{attribute 'linkalways'} 
{attribute 'no_explicit_call' := 'This FB is a CLASS and must be accessed using methods or properties'}
{attribute 'enable_dynamic_creation'}
FUNCTION_BLOCK _ETcVnFeatureScalingType EXTENDS EnumDatatypeBase
VAR
	localData : ETcVnFeatureScalingType;
	activeData : REFERENCE TO ETcVnFeatureScalingType;
	enumBaseDatatype : _DINT(localData);
END_VAR

METHOD PRIVATE AddLocalEnumeration
VAR_INPUT
	Enumeration : T_MAXSTRING;
	Value : ETcVnFeatureScalingType;
END_VAR
AddEnumeration(Enumeration, Value);
END_METHOD

PROPERTY PUBLIC Address : PVOID
GET
Address := ADR(activeData);
END_GET
END_PROPERTY

METHOD PUBLIC ClearReference
VAR_INPUT
END_VAR
activeData REF= localData;
SetBaseDatatypeReference();
END_METHOD

METHOD PUBLIC Clone : I_Datatype
VAR
    pClone : POINTER TO _ETcVnFeatureScalingType;
END_VAR
pClone := __NEW(_ETcVnFeatureScalingType(InitialValue := Value));
Clone := pClone^;
END_METHOD

METHOD FB_init : BOOL
VAR_INPUT
	bInitRetains : BOOL; // if TRUE, the retain variables are initialized (warm start / cold start)
	bInCopyCode : BOOL;  // if TRUE, the instance afterwards gets moved into the copy code (online change)
	InitialValue : ETcVnFeatureScalingType;
END_VAR
localData := InitialValue;
AddBaseDatatype(enumBaseDatatype);
ClearReference();

AddLocalEnumeration('TCVN_FST1_MAXABS', ETcVnFeatureScalingType.TCVN_FST1_MAXABS);
AddLocalEnumeration('TCVN_FST1_MINMAX', ETcVnFeatureScalingType.TCVN_FST1_MINMAX);
AddLocalEnumeration('TCVN_FST1_STANDARDIZATION', ETcVnFeatureScalingType.TCVN_FST1_STANDARDIZATION);
END_METHOD

PROPERTY PUBLIC Identifier : T_MAXSTRING
GET
Identifier := 'ETcVnFeatureScalingType';
END_GET
END_PROPERTY

METHOD IsEnumeratorValueEqual : BOOL
VAR_INPUT
	Enumerator : I_KeyValueForwardEnumerator;
END_VAR
VAR
	storedValue : ETcVnFeatureScalingType;
END_VAR
IF NOT Enumerator.TryGet(storedValue) THEN
	RETURN;
END_IF

IsEnumeratorValueEqual := storedValue = activeData;
END_METHOD

METHOD PUBLIC MakeReferenceTo
VAR_INPUT
	ReferenceTarget : REFERENCE TO ETcVnFeatureScalingType;
END_VAR
activeData REF= ReferenceTarget;
SetBaseDatatypeReference();
END_METHOD

METHOD PROTECTED SetBaseDatatypeReference
VAR_INPUT
END_VAR
enumBaseDatatype.MakeReferenceTo(activeData);
END_METHOD

PROPERTY PUBLIC Size : UDINT
GET
Size := SIZEOF(activeData);
END_GET
END_PROPERTY

METHOD TryMakeReferenceTo : BOOL
VAR_INPUT
	Target : I_Datatype;
END_VAR
VAR
	targetAsEnum : I_EnumDatatype;
	pTargetData : POINTER TO ETcVnFeatureScalingType;
END_VAR
IF NOT Target.TryResolveAsEnumDatatype(targetAsEnum) THEN
	RETURN;
END_IF

IF targetAsEnum.Identifier <> Identifier THEN
	RETURN;
END_IF

pTargetData := Target.Address;
activeData REF= pTargetData^;
SetBaseDatatypeReference();
TryMakeReferenceTo := TRUE;
END_METHOD

PROPERTY PUBLIC Value : ETcVnFeatureScalingType
GET
Value := activeData;
END_GET
SET
activeData := Value;
END_SET
END_PROPERTY

END_FUNCTION_BLOCK

(* stored: Version 1.1.0.1
   POU _ETcVnFeatureScalingType: Id {cbdc24b0-4f4a-49ca-9aec-b0942f16fccc}, SpecialFunc None
   Folder Constructor: Id {c77c6d3e-50f5-4cd6-991a-3f0ec9075f30}
   Folder Private: Id {1b0b0be0-4d66-47cd-9a6e-5487d0e514bd}
   Folder Protected: Id {7a90c783-6383-4e35-afdc-7b29e1d37f08}
   Method AddLocalEnumeration: Id {a2e2968b-13c1-468c-add2-f94a5ca75525}
   Property Address: Id {d03bf062-f79f-4257-b84c-9fd60c486463}
   Get Get: Id {0546e3ee-fefc-472c-8471-374989596c6b}
   Method ClearReference: Id {024ec11e-01ca-419a-981c-1df142e831a0}
   Method Clone: Id {614bb093-8beb-4ecf-ae74-1470c7cc00e3}
   Method FB_init: Id {aa75cf16-16d4-4e58-8503-10a44bda474a}
   Property Identifier: Id {a724169f-08d5-435c-98d9-90c313dbc9d7}
   Get Get: Id {8f9012fd-5594-4cee-9437-22cf5db2703b}
   Method IsEnumeratorValueEqual: Id {1371d5c2-abb3-4db5-a72f-aacea151a3c8}
   Method MakeReferenceTo: Id {577521bf-75bc-4bf7-9095-611abd96db03}
   Method SetBaseDatatypeReference: Id {92d24912-f955-4f7c-871d-74baea4ae771}
   Property Size: Id {f36c3807-b7b3-4dab-9b65-18dc6710b258}
   Get Get: Id {e8639ba0-3c3e-4e16-94fa-b3c7489cf03a}
   Method TryMakeReferenceTo: Id {cd12e511-9400-4404-a2fe-eada058473c6}
   Property Value: Id {0b7584af-13ad-499f-afed-455720f6ac7c}
   Get Get: Id {96ad0bd7-615a-4346-8bd7-e1233b2f499f}
   Set Set: Id {a7a7ac56-2bca-4da8-9f65-f9d6d412d46d} *)
